// Struckig
// Copyright (C) 2022 Stefan Besler

// This program is free software: you can redistribute it and/or modify
// it under the terms of the GNU General Public License as published by
// the Free Software Foundation, either version 3 of the License, or
// (at your option) any later version.

// This program is distributed in the hope that it will be useful,
// but WITHOUT ANY WARRANTY; without even the implied warranty of
// MERCHANTABILITY or FITNESS FOR A PARTICULAR PURPOSE.  See the
// GNU General Public License for more details.
//
// You should have received a copy of the GNU General Public License
// along with THIS PROGRAM.  IF NOT, see <http://www.gnu.org/licenses/>.
/// Which times are possible for synchronization?
TYPE INTERNAL BlockInterval :
STRUCT
  IsUsed : BOOL;
  Left, Right : LREAL;
  Profile : ProfileDesc;
END_STRUCT
END_TYPE

(* stored: Version 1.1.0.1
   DUT BlockInterval: Id {ddb6295e-c8fd-4ec6-9011-9c80b2d7a348} *)
